FUNCTION_BLOCK Ramp
VAR_INPUT
END_VAR
VAR_OUTPUT
	m_presenceSensorRampFull : PresenceSensor;
END_VAR
VAR
END_VAR

END_FUNCTION_BLOCK

(* stored: Version 1.1.0.1, ProductVersion 3.1.4024.4
   POU Ramp: Id {17692bb4-989c-44d5-827a-7486b12de95c}, SpecialFunc None *)
